// TIA Portal V16 program export: 2 tag tables, 0 data types, 1 data blocks, 1 code blocks (in call order from the OBs), 6 instance data blocks

VAR_GLOBAL   // PLC tag table "Default tag table"
   STOP AT %M0.0 : Bool;
   START AT %M0.1 : Bool;
   "READY 2 Run" AT %M0.2 : Bool;
   "Actual pcs" AT %MW2 : Int;
   "Another Piece" AT %M0.3 : Bool;
   "Full Box" AT %M0.4 : Bool;
   PulseFlag AT %M0.5 : Bool;
   PulseOut AT %M0.6 : Bool;
   "Box Capacity" AT %MW8 : Int;
   "Sensor Final" AT %M1.2 : Bool;
   "Sensor Middle" AT %M1.1 : Bool;
   "Sensor Start" AT %M1.0 : Bool;
   "Pcs in Extrusion" AT %MW4 : Int;
   "Extrusions in Box" AT %MW6 : Int;
   "Actual extrusion" AT %MW10 : Int;
   "Coveyor 2 Delay" AT %MD12 : Time;
END_VAR
VAR_GLOBAL CONSTANT   // user constants
   "Krabica mala" : Int := 150;
   "Krabica velka" : Int := 250;
END_VAR

VAR_GLOBAL   // PLC tag table "Input & Output table"
   "Conveyor 1" AT %Q0.0 : Bool;
   "Conveyor 2" AT %Q0.1 : Bool;
   Green AT %Q0.2 : Bool;
   Yellow AT %Q0.3 : Bool;
   Red AT %Q0.4 : Bool;
END_VAR

DATA_BLOCK "HMI Communication"   // DB7
{ S7_Optimized_Access := 'TRUE' }
VERSION : 0.1
// stored: AutoNumber true, DBAccessibleFromOPCUA true, IsOnlyStoredInLoadMemory false, IsRetainMemResEnabled false, IsWriteProtectedInAS false, MemoryReserve 100
   VAR
      "Sensor Final" : Bool;
      "Sensor Middle" : Bool;
      "Sensor Start" : Bool;
   END_VAR
BEGIN
END_DATA_BLOCK

ORGANIZATION_BLOCK "Main"   // OB1, LAD, ProgramCycle
TITLE = "Main Program Sweep (Cycle)"
{ S7_Optimized_Access := 'TRUE' }
VERSION : 0.1
// stored: AutoNumber true, IsIECCheckEnabled false, SetENOAutomatically false
   VAR_INPUT
      Initial_Call : Bool;   // Initial call of this OB
      Remanence : Bool;   // =True, if remanent data are available
   END_VAR
   VAR CONSTANT
      start : Bool;
   END_VAR
BEGIN

REGION Network 1: Spustenie a zastavenie automatického režimu
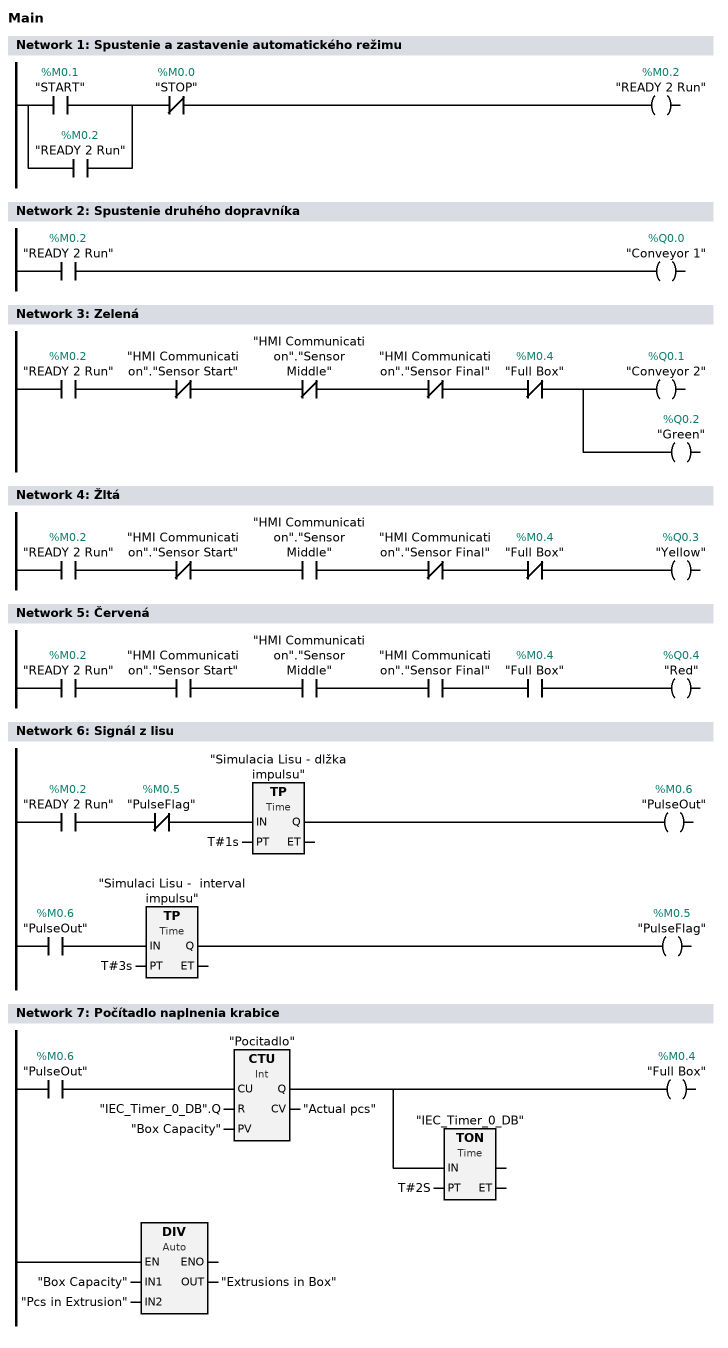
   RUNG wire#powerrail
      Contact( "START" )
      wire#w1
      I_Contact( "STOP" )
      Coil( "READY 2 Run" )
   END_RUNG
   RUNG wire#powerrail
      Contact( "READY 2 Run" )
   END_RUNG wire#w1
   // the same network as SCL:
   "READY 2 Run" := ("START" OR "READY 2 Run") AND NOT "STOP";
END_REGION

REGION Network 2: Spustenie druhého dopravníka
   RUNG wire#powerrail
      Contact( "READY 2 Run" )
      Coil( "Conveyor 1" )
   END_RUNG
   // the same network as SCL:
   "Conveyor 1" := "READY 2 Run";
END_REGION

REGION Network 3: Zelená
   RUNG wire#powerrail
      Contact( "READY 2 Run" )
      I_Contact( "HMI Communication"."Sensor Start" )
      I_Contact( "HMI Communication"."Sensor Middle" )
      I_Contact( "HMI Communication"."Sensor Final" )
      I_Contact( "Full Box" )
      wire#w1
      Coil( "Conveyor 2" )
   END_RUNG
   RUNG wire#w1
      Coil( "Green" )
   END_RUNG
   // the same network as SCL:
   "Conveyor 2" := "READY 2 Run" AND NOT "HMI Communication"."Sensor Start" AND NOT "HMI Communication"."Sensor Middle" AND NOT "HMI Communication"."Sensor Final" AND NOT "Full Box";
   "Green" := "Conveyor 2";
END_REGION

REGION Network 4: Žltá
   RUNG wire#powerrail
      Contact( "READY 2 Run" )
      I_Contact( "HMI Communication"."Sensor Start" )
      Contact( "HMI Communication"."Sensor Middle" )
      I_Contact( "HMI Communication"."Sensor Final" )
      I_Contact( "Full Box" )
      Coil( "Yellow" )
   END_RUNG
   // the same network as SCL:
   "Yellow" := "READY 2 Run" AND NOT "HMI Communication"."Sensor Start" AND "HMI Communication"."Sensor Middle" AND NOT "HMI Communication"."Sensor Final" AND NOT "Full Box";
END_REGION

REGION Network 5: Červená
   RUNG wire#powerrail
      Contact( "READY 2 Run" )
      Contact( "HMI Communication"."Sensor Start" )
      Contact( "HMI Communication"."Sensor Middle" )
      Contact( "HMI Communication"."Sensor Final" )
      Contact( "Full Box" )
      Coil( "Red" )
   END_RUNG
   // the same network as SCL:
   "Red" := "READY 2 Run" AND "HMI Communication"."Sensor Start" AND "HMI Communication"."Sensor Middle" AND "HMI Communication"."Sensor Final" AND "Full Box";
END_REGION

REGION Network 6: Signál z lisu
   RUNG wire#powerrail
      Contact( "READY 2 Run" )
      I_Contact( "PulseFlag" )
      { S7_Templates := "time_type := Time" } "Simulacia Lisu - dlžka impulsu".TP(pt := T#1s, et =>)
      Coil( "PulseOut" )
   END_RUNG
   RUNG wire#powerrail
      Contact( "PulseOut" )
      { S7_Templates := "time_type := Time" } "Simulaci Lisu -  interval impulsu".TP(pt := T#3s, et =>)
      Coil( "PulseFlag" )
   END_RUNG
   // the same network as SCL:
   "Simulacia Lisu - dlžka impulsu".TP(IN := "READY 2 Run" AND NOT "PulseFlag", PT := T#1s);
   "PulseOut" := "Simulacia Lisu - dlžka impulsu".Q;
   "Simulaci Lisu -  interval impulsu".TP(IN := "PulseOut", PT := T#3s);
   "PulseFlag" := "Simulaci Lisu -  interval impulsu".Q;
END_REGION

REGION Network 7: Počítadlo naplnenia krabice
   RUNG wire#powerrail
      Contact( "PulseOut" )
      { S7_Templates := "value_type := Int" } "Pocitadlo".CTU(r := "IEC_Timer_0_DB".Q, pv := "Box Capacity", cv => "Actual pcs")
      wire#w1
      Coil( "Full Box" )
   END_RUNG
   RUNG wire#w1
      { S7_Templates := "time_type := Time" } "IEC_Timer_0_DB".TON(pt := T#2S, et =>)
   END_RUNG
   RUNG wire#powerrail
      Div(in1 := "Box Capacity", in2 := "Pcs in Extrusion", out => "Extrusions in Box")
   END_RUNG
   // the same network as SCL:
   "Pocitadlo".CTU(CU := "PulseOut", R := "IEC_Timer_0_DB".Q, PV := "Box Capacity", CV => "Actual pcs");
   "Full Box" := "Pocitadlo".Q;
   "IEC_Timer_0_DB".TON(IN := "Pocitadlo".Q, PT := T#2S);
   "Extrusions in Box" := "Box Capacity" / "Pcs in Extrusion";
END_REGION
END_ORGANIZATION_BLOCK

DATA_BLOCK "IEC_Counter_0_DB"   // DB2
{ S7_Optimized_Access := 'TRUE' }
// stored: AutoNumber true, DBAccessibleFromOPCUA true, InstanceOfName IEC_COUNTER, OfSystemLibElement IEC_COUNTER, OfSystemLibVersion 1.0
"IEC_COUNTER"
   // VAR RETAIN
   //    CU : Bool;
   //    CD : Bool;
   //    R : Bool;
   //    LD : Bool;
   //    QU : Bool;
   //    QD : Bool;
   //    PV : Int;
   //    CV : Int;
   // END_VAR
BEGIN
END_DATA_BLOCK

DATA_BLOCK "IEC_Timer_0_DB"   // DB5
{ S7_Optimized_Access := 'TRUE' }
// stored: AutoNumber true, DBAccessibleFromOPCUA true, InstanceOfName IEC_TIMER, OfSystemLibElement IEC_TIMER, OfSystemLibVersion 1.0
"IEC_TIMER"
   // VAR
   //    PT : Time;
   //    ET { ExternalWritable := 'False'} : Time;
   //    IN : Bool;
   //    Q { ExternalWritable := 'False'} : Bool;
   // END_VAR
BEGIN
END_DATA_BLOCK

DATA_BLOCK "Pocitadlo"   // DB6
{ S7_Optimized_Access := 'TRUE' }
// stored: AutoNumber true, DBAccessibleFromOPCUA true, InstanceOfName IEC_COUNTER, OfSystemLibElement IEC_COUNTER, OfSystemLibVersion 1.0
"IEC_COUNTER"
   // VAR RETAIN
   //    CU : Bool;
   //    CD : Bool;
   //    R : Bool;
   //    LD : Bool;
   //    QU : Bool;
   //    QD : Bool;
   //    PV : Int;
   //    CV : Int;
   // END_VAR
BEGIN
END_DATA_BLOCK

DATA_BLOCK "Simulaci Lisu -  interval impulsu"   // DB3
{ S7_Optimized_Access := 'TRUE' }
// stored: AutoNumber true, DBAccessibleFromOPCUA true, InstanceOfName IEC_TIMER, OfSystemLibElement IEC_TIMER, OfSystemLibVersion 1.0
"IEC_TIMER"
   // VAR
   //    PT : Time;
   //    ET { ExternalWritable := 'False'} : Time;
   //    IN : Bool;
   //    Q { ExternalWritable := 'False'} : Bool;
   // END_VAR
BEGIN
END_DATA_BLOCK

DATA_BLOCK "Simulacia Lisu - dlžka impulsu"   // DB4
{ S7_Optimized_Access := 'TRUE' }
// stored: AutoNumber true, DBAccessibleFromOPCUA true, InstanceOfName IEC_TIMER, OfSystemLibElement IEC_TIMER, OfSystemLibVersion 1.0
"IEC_TIMER"
   // VAR
   //    PT : Time;
   //    ET { ExternalWritable := 'False'} : Time;
   //    IN : Bool;
   //    Q { ExternalWritable := 'False'} : Bool;
   // END_VAR
BEGIN
END_DATA_BLOCK

DATA_BLOCK "Simulácia Lisu"   // DB1
{ S7_Optimized_Access := 'TRUE' }
// stored: AutoNumber true, DBAccessibleFromOPCUA true, InstanceOfName IEC_TIMER, OfSystemLibElement IEC_TIMER, OfSystemLibVersion 1.0
"IEC_TIMER"
   // VAR
   //    PT : Time;
   //    ET { ExternalWritable := 'False'} : Time;
   //    IN : Bool;
   //    Q { ExternalWritable := 'False'} : Bool;
   // END_VAR
BEGIN
END_DATA_BLOCK
